// TIA Portal V17 export
// export: Created 2024-09-03T21:54:51.7361873Z, ExportSetting WithDefaults, DisplayName Totally Integrated Automation Portal, DisplayVersion V17 Update 7, DisplayName TIA Portal Openness, DisplayVersion V17 Update 7, DisplayName TIA Portal Version Control Interface, DisplayVersion V17, DisplayName SINAMICS Startdrive Advanced, DisplayVersion V17 SP2, DisplayName SINAMICS Startdrive G110M, G120, G120C, G120D, G120P, G115D, DisplayVersion V17 SP2, DisplayName SINAMICS Startdrive G130, G150, S120, S150, SINAMICS MV, S210, DisplayVersion V17 SP2, DisplayName STEP 7 Professional, DisplayVersion V17 Update 7, DisplayName STEP 7 Safety, DisplayVersion V17 Update 6, DisplayName WinCC Advanced / Unified PC, DisplayVersion V17 Update 7
DATA_BLOCK "Manipulator_main_DB"   // DB42
VERSION : 0.1
// stored: AutoNumber true, DBAccessibleFromOPCUA true, DBAccessibleFromWebserver true, InstanceOfName Manipulator_main, InstanceOfType FB
"Manipulator_main"
   // VAR
   //    PUT_Instance : PUT;
   //    GET_Instance : GET;
   //    GetStatusMem : Word;
   //    PutStatusMem : Word;
   //    GetCounterNDR : ULInt;
   //    PutCounterDone : ULInt;
   //    GetCounterNDR_last : ULInt;
   //    PutCounterDone_last : ULInt;
   //    GetCommOK : Bool;
   //    PutCommOK : Bool;
   //    R_TRIG_GetNDR : R_TRIG;
   //    R_TRIG_PutDone : R_TRIG;
   //    IEC_Timer_GetCommOK { S7_SetPoint := 'True'} : TOF_TIME;
   //    IEC_Timer_PutCommOK { S7_SetPoint := 'True'} : TOF_TIME;
   // END_VAR
BEGIN
END_DATA_BLOCK
